FUNCTION_BLOCK FB_StateBegin IMPLEMENTS I_State
VAR
	_refMainStateMachine		: REFERENCE TO FB_MainStateMachine;
	_fbTcMessage				: FB_TcMessage;
	_fbTon						: TON;
END_VAR

METHOD SafetyTripped
VAR_INPUT
END_VAR
END_METHOD

METHOD FB_init : BOOL
VAR_INPUT
	// if TRUE, the retain variables are initialized (warm start / cold start)
	bInitRetains			: BOOL;
	// if TRUE, the instance afterwards gets moved into the copy code (online
	// change)
	bInCopyCode				: BOOL;
	fbMainStateMachine		: REFERENCE TO FB_MainStateMachine;
END_VAR
_refMainStateMachine REF= fbMainStateMachine;
_fbTcMessage.CreateEx(
	stEventEntry	:= TC_EVENTS.StatePatternEvents.Info001MachineStarted,
	ipSourceInfo	:= 0);
END_METHOD

METHOD SafetyAcknowledged
VAR_INPUT
END_VAR
END_METHOD

METHOD ClearErrors
END_METHOD

METHOD StartButtonPressed
END_METHOD

METHOD GetDescription : STRING
GetDescription := 'Begin';
END_METHOD

METHOD Execute
IF _TaskInfo[GETCURTASKINDEXEX()].FirstCycle THEN
	_fbTcMessage.Send(0);
END_IF

_fbTon(IN := TRUE, PT := T#100MS);

IF _fbTon.Q THEN
	_fbTon(IN := FALSE);
	_refMainStateMachine.SetState(_refMainStateMachine.ipStateReadParameters);
END_IF
END_METHOD

METHOD StopButtonPressed
END_METHOD

END_FUNCTION_BLOCK

(* stored: Version 1.1.0.1, ProductVersion 3.1.4024.11
   POU FB_StateBegin: Id {c23222e7-7a85-4c4b-a6b1-9f625840daab}, SpecialFunc None
   Method SafetyTripped: Id {277a61e6-9929-4cb6-aa21-37cab37b30b1}
   Method FB_init: Id {33555ac9-e0a1-4814-a475-2455dfbd8bc2}
   Method SafetyAcknowledged: Id {4f3eaf11-4b9a-40d6-90b6-54949ff4e956}
   Method ClearErrors: Id {6a44044f-3ac7-4935-b041-5a34f290078f}
   Method StartButtonPressed: Id {b6a0d132-31af-496e-98eb-7e72428faef5}
   Method GetDescription: Id {cebf82b6-8992-45d1-95c0-240ff92b556d}
   Method Execute: Id {e5d4d2b8-6c9c-41f9-9f36-2371c8c34bae}
   Method StopButtonPressed: Id {fc92dfe7-ccb9-4be4-b335-3eaf6b74bcbc} *)
